TYPE Reactor EXTENDS Vessel :
STRUCT
	TemperatureInputRaw : INT;
	PressureInputRaw : INT;
	LevelInputRaw : INT;
	
	VFD : VFD;
END_STRUCT
END_TYPE

(* stored: Version 1.1.0.1, ProductVersion 3.1.4024.3
   DUT Reactor: Id {06bb757a-a2f8-407e-a9eb-320344b48588} *)
